(* IEC 61131-3 sources: Word/plc-course/16-alarms-and-diagnostics/labs/starter, 3 files *)

(* ---- 16-1-alarm-block.st ---- *)
(* Lab 16-1: FB_Alarm - one alarm with an on-delay, optional latching,
   edge-triggered acknowledge and reset, and the alarm states an HMI needs.
   Module 16 (Alarms, diagnostics and fault handling). STARTER - the state
   type, the block interface and the program that uses the block are done
   for you; write the body of FB_Alarm where it says TODO, then run:
     python3 tools/plctest.py 16-alarms-and-diagnostics/labs/starter/16-1-alarm-block.st

   Tips: keep Active and Unacked as two separate memories and derive State
   from them at the end. Think about the ORDER of acknowledge and
   activation inside one scan. *)

TYPE
  E_AlarmState : (
    Normal,        (* not active, nothing to acknowledge *)
    ActiveUnack,   (* active, not yet acknowledged: flash + horn *)
    ActiveAcked,   (* active, acknowledged, condition still present: steady *)
    RtnUnack,      (* returned to normal before anyone acknowledged it *)
    LatchedRtn     (* latching alarm: acknowledged, condition gone, waiting for reset *)
  );
END_TYPE

FUNCTION_BLOCK FB_Alarm
  VAR_INPUT
    Condition : BOOL;   (* raw alarm condition from the process logic *)
    OnDelay   : TIME;   (* Condition must last this long before the alarm activates *)
    Latching  : BOOL;   (* TRUE: stays active after the condition clears, until Reset *)
    Ack       : BOOL;   (* acknowledge command: acts on its rising edge *)
    Reset     : BOOL;   (* reset command for a latching alarm: acts on its rising edge *)
  END_VAR
  VAR_OUTPUT
    Active    : BOOL;   (* alarm is active: confirmed condition, or latched *)
    Unacked   : BOOL;   (* the latest activation has not been acknowledged *)
    State     : E_AlarmState;
    Count     : DINT;   (* activations since power-up, for alarm statistics *)
  END_VAR
  VAR
    (* Add your internal variables here (timer, edge detectors ...). *)
    DelayTimer : TON;
  END_VAR

  (* TODO: replace these placeholder lines with your logic (see the
     requirements in the Module 16 README, Lab 16-1). *)
  Active := FALSE;
  Unacked := FALSE;
  State := Normal;
  Count := 0;
END_FUNCTION_BLOCK

PROGRAM AlarmDemo
  VAR (* panel push-buttons and horn *)
    AckPB   AT %IX0.0 : BOOL;   (* Acknowledge push-button, NO *)
    ResetPB AT %IX0.1 : BOOL;   (* Reset push-button, NO *)
    Horn    AT %QX0.0 : BOOL;   (* Alarm horn *)
  END_VAR
  VAR (* alarm conditions: in a real program they come from process logic
         (for example FB_AnalogAlarm, Lab 14-2). Here the test writes them. *)
    TempHigh : BOOL;   (* TT-201 compressor bearing temperature high *)
    VibHigh  : BOOL;   (* VT-202 compressor vibration high-high *)
    DoorOpen : BOOL;   (* acoustic enclosure door open *)
  END_VAR
  VAR
    TempAlm : FB_Alarm;
    VibAlm  : FB_Alarm;
    DoorAlm : FB_Alarm;
  END_VAR

  (* The program is complete: do not change these calls. *)
  TempAlm(Condition := TempHigh, OnDelay := T#3s, Latching := FALSE, Ack := AckPB, Reset := ResetPB);
  VibAlm(Condition := VibHigh, OnDelay := T#1s, Latching := TRUE, Ack := AckPB, Reset := ResetPB);
  DoorAlm(Condition := DoorOpen, OnDelay := T#0s, Latching := FALSE, Ack := AckPB, Reset := ResetPB);

  (* The horn sounds while any alarm is unacknowledged. *)
  Horn := TempAlm.Unacked OR VibAlm.Unacked OR DoorAlm.Unacked;
END_PROGRAM

CONFIGURATION Config0
  RESOURCE Res0 ON PLC
    TASK MainTask(INTERVAL := T#10ms, PRIORITY := 0);
    PROGRAM Inst0 WITH MainTask : AlarmDemo;
  END_RESOURCE
END_CONFIGURATION

(* ---- 16-3-frozen-signal-heartbeat.st ---- *)
(* Lab 16-3: Frozen-signal and heartbeat diagnostics.
   Module 16 (Alarms, diagnostics and fault handling). STARTER - the block
   interfaces and the program that uses them are done for you. Write:
     1. the body of FB_FrozenSignal,
     2. the body of FB_Heartbeat,
     3. this PLC's own heartbeat (HeartbeatOut) at the end of the program,
   where it says TODO, then run:
     python3 tools/plctest.py 16-alarms-and-diagnostics/labs/starter/16-3-frozen-signal-heartbeat.st

   Two small diagnostic blocks that catch faults a range check cannot see:
     FB_FrozenSignal  a transmitter value that stops moving while the
                      process is running (stuck sensor, transmitter left in
                      fixed-current mode, frozen communication value)
     FB_Heartbeat     a partner's heartbeat counter that stops changing
                      (partner stopped, or the link between us is down) *)

FUNCTION_BLOCK FB_FrozenSignal
  VAR_INPUT
    PV         : REAL;   (* value to watch, engineering units *)
    Tolerance  : REAL;   (* a change larger than this counts as movement *)
    FreezeTime : TIME;   (* no movement for this long = frozen *)
    Enable     : BOOL;   (* TRUE while the process should make PV move *)
  END_VAR
  VAR_OUTPUT
    Frozen     : BOOL;   (* PV has not moved by more than Tolerance for FreezeTime *)
  END_VAR
  VAR
    (* Add your internal variables here. Hint: compare PV with a REFERENCE
       value, not with the previous scan's value. *)
    StillTimer : TON;
  END_VAR

  (* TODO: replace this placeholder line with your logic (see the
     requirements in the Module 16 README, Lab 16-3). *)
  Frozen := FALSE;
END_FUNCTION_BLOCK

FUNCTION_BLOCK FB_Heartbeat
  VAR_INPUT
    Counter   : INT;     (* heartbeat counter received from the partner *)
    Timeout   : TIME;    (* no change for this long = partner or link lost *)
  END_VAR
  VAR_OUTPUT
    CommOK    : BOOL;    (* partner proven alive within the last Timeout *)
    CommFault : BOOL;    (* no change for Timeout: raise an alarm *)
  END_VAR
  VAR
    (* Add your internal variables here. *)
    SilentTimer : TON;
  END_VAR

  (* TODO: replace these placeholder lines with your logic. *)
  CommOK := FALSE;
  CommFault := FALSE;
END_FUNCTION_BLOCK

PROGRAM PumpDiagnostics
  VAR (* I/O *)
    PumpRunFb AT %IX0.0 : BOOL;   (* P-301 contactor auxiliary contact: TRUE = running *)
    FrozenAlm AT %QX0.0 : BOOL;   (* a transmitter looks frozen *)
    CommAlm   AT %QX0.1 : BOOL;   (* a heartbeat has been lost *)
  END_VAR
  VAR (* values from the analog input blocks (Lab 14-1) and the communication
         driver (Module 17). Here the test writes them directly. *)
    PT301        : REAL;   (* P-301 discharge pressure, bar *)
    FT302        : REAL;   (* P-301 discharge flow, m3/h *)
    PartnerHB    : INT;    (* heartbeat counter from PLC-2: it adds 1 every second *)
    ScadaHB      : INT;    (* watchdog counter the SCADA server writes every few seconds *)
    HeartbeatOut : INT;    (* this PLC's own heartbeat, read by PLC-2 and SCADA *)
  END_VAR
  VAR
    PT301Chk   : FB_FrozenSignal;
    FT302Chk   : FB_FrozenSignal;
    PartnerMon : FB_Heartbeat;
    ScadaMon   : FB_Heartbeat;
    (* add a timer for HeartbeatOut here *)
  END_VAR

  (* The calls below are complete: do not change them.
     A running pump's discharge pressure and flow always move a little
     (pulsation, turbulence). When the pump is stopped they may be dead
     steady, so the check only runs while the pump runs. *)
  PT301Chk(PV := PT301, Tolerance := 0.05, FreezeTime := T#10s, Enable := PumpRunFb);
  FT302Chk(PV := FT302, Tolerance := 0.5, FreezeTime := T#20s, Enable := PumpRunFb);

  (* PLC-2 counts once a second: 3 s allows two missed updates.
     SCADA writes more slowly and less regularly: 10 s. *)
  PartnerMon(Counter := PartnerHB, Timeout := T#3s);
  ScadaMon(Counter := ScadaHB, Timeout := T#10s);

  FrozenAlm := PT301Chk.Frozen OR FT302Chk.Frozen;
  CommAlm := PartnerMon.CommFault OR ScadaMon.CommFault;

  (* TODO: this PLC's own heartbeat. HeartbeatOut starts at 0 and adds 1
     every second; after 32767 it goes back to 0. Replace the placeholder. *)
  HeartbeatOut := 0;
END_PROGRAM

CONFIGURATION Config0
  RESOURCE Res0 ON PLC
    TASK MainTask(INTERVAL := T#10ms, PRIORITY := 0);
    PROGRAM Inst0 WITH MainTask : PumpDiagnostics;
  END_RESOURCE
END_CONFIGURATION

(* ---- 16-2-first-out-annunciator.st ---- *)
(* Lab 16-2: First-out annunciator for the eight shutdown inputs of a gas
   compressor, with horn, acknowledge, reset, lamp test and a run permissive.
   Module 16 (Alarms, diagnostics and fault handling). STARTER - the I/O and
   the HMI status arrays are declared for you; write the logic where it says
   TODO, then run:
     python3 tools/plctest.py 16-alarms-and-diagnostics/labs/starter/16-2-first-out-annunciator.st

   TRAINING EXERCISE ONLY: on a real compressor the shutdown function itself
   belongs in a properly designed (often safety-rated) trip system. This lab
   is about annunciation: showing the operator what tripped, and what
   tripped FIRST.

   Tip: copy the eight inputs into a BOOL array first, then every rule
   becomes a FOR loop over the channels. Decide carefully in which ORDER
   the steps run inside one scan. *)

PROGRAM FirstOutPanel
  VAR (* trip inputs: NC contacts, TRUE = healthy, FALSE = tripped or wire broken *)
    Trip1_NC   AT %IX0.0 : BOOL;  (* PSLL-401 suction pressure low-low *)
    Trip2_NC   AT %IX0.1 : BOOL;  (* PSHH-402 discharge pressure high-high *)
    Trip3_NC   AT %IX0.2 : BOOL;  (* TSHH-403 discharge temperature high-high *)
    Trip4_NC   AT %IX0.3 : BOOL;  (* PSLL-404 lube oil pressure low-low *)
    Trip5_NC   AT %IX0.4 : BOOL;  (* VSHH-405 vibration high-high *)
    Trip6_NC   AT %IX0.5 : BOOL;  (* LSHH-406 suction scrubber level high-high *)
    Trip7_NC   AT %IX0.6 : BOOL;  (* HS-407 local shutdown push-button (monitoring contact) *)
    Trip8_NC   AT %IX0.7 : BOOL;  (* XA-408 main motor protection relay trip *)
    AckPB      AT %IX1.0 : BOOL;  (* Acknowledge (silence) push-button, NO *)
    ResetPB    AT %IX1.1 : BOOL;  (* Reset push-button, NO *)
    LampTestPB AT %IX1.2 : BOOL;  (* Lamp test push-button, NO *)
    Lamp1      AT %QX0.0 : BOOL;  (* annunciator window lamps, one per channel *)
    Lamp2      AT %QX0.1 : BOOL;
    Lamp3      AT %QX0.2 : BOOL;
    Lamp4      AT %QX0.3 : BOOL;
    Lamp5      AT %QX0.4 : BOOL;
    Lamp6      AT %QX0.5 : BOOL;
    Lamp7      AT %QX0.6 : BOOL;
    Lamp8      AT %QX0.7 : BOOL;
    Horn       AT %QX1.0 : BOOL;  (* audible alarm *)
    RunPermit  AT %QX1.1 : BOOL;  (* TRUE = compressor may be started (no channel latched) *)
  END_VAR
  VAR (* status for the HMI, one element per channel *)
    Latched  : ARRAY[1..8] OF BOOL;  (* channel has tripped and has not been reset *)
    Unacked  : ARRAY[1..8] OF BOOL;  (* channel trip not yet acknowledged *)
    FirstOut : ARRAY[1..8] OF BOOL;  (* channel was (one of) the first to trip *)
  END_VAR
  VAR
    (* Add your internal variables here (arrays, edge detectors, flasher ...). *)
    I : INT;
  END_VAR

  (* TODO: replace these placeholder lines with your logic (see the
     requirements in the Module 16 README, Lab 16-2). *)
  Lamp1 := FALSE;
  Lamp2 := FALSE;
  Lamp3 := FALSE;
  Lamp4 := FALSE;
  Lamp5 := FALSE;
  Lamp6 := FALSE;
  Lamp7 := FALSE;
  Lamp8 := FALSE;
  Horn := FALSE;
  RunPermit := FALSE;
END_PROGRAM

CONFIGURATION Config0
  RESOURCE Res0 ON PLC
    TASK MainTask(INTERVAL := T#10ms, PRIORITY := 0);
    PROGRAM Inst0 WITH MainTask : FirstOutPanel;
  END_RESOURCE
END_CONFIGURATION
